PROGRAM Alarm
VAR
	Timer_allarme: TON;
	allarme_tamper:BOOL;
	Timer_Sirena: TP;
	alarm_service: BOOL;
	rilevato_movimento: BOOL;
	rilevata_manomissione: BOOL;
	allarme_scattato: BOOL;
	SR_ainterno: SR;
	SR_afronte: SR;
	SR_aretro: SR;
	SR_asx: SR;
	SR_allarme: SR;
	SR_atamper: SR;
	SR_mensa: SR;
	SR_ingresso: SR;
	SR_tecnico: SR;
	
	F1_trig: F_TRIG;
	F2_trig: F_TRIG;
	F3_trig: F_TRIG;
	F4_trig: F_TRIG;
	F5_trig: F_TRIG;
	S1_trig: F_TRIG;
	S2_trig: F_TRIG;
	R1_trig: F_TRIG;
	R2_trig: F_TRIG;
	R3_trig: F_TRIG;
	R4_trig: F_TRIG;
	R5_trig: F_TRIG;
	D1_trig: F_TRIG;
	C1_trig: F_TRIG;
	C2_trig: F_TRIG;
	C3_trig: F_TRIG;
	U1_trig: F_TRIG;
	U2_trig: F_TRIG;
	U3_trig: F_TRIG;

	F1_count: INT;
	F2_count: INT;
	F3_count: INT;
	F4_count: INT;
	F5_count: INT;
	S1_count: INT;
	S2_count: INT;
	R1_count: INT;
	R2_count: INT;
	R3_count: INT;
	R4_count: INT;
	R5_count: INT;
	D1_count: INT;
	C1_count: INT;
	C2_count: INT;
	C3_count: INT;
	U1_count: INT;
	U2_count: INT;
	U3_count: INT;
	radio_count: INT;
	sirena_count: INT;
	allarm_trig: R_TRIG;
	rtrig_radio: R_TRIG;
	rtrig_sirena: R_TRIG;
END_VAR

act();
(*Ritardo avvio allarme su accensione*)
//Timer_allarme(IN:= allarme, PT:= delay_allarme_on, Q=> allarme_on, ET=> );
(*Sensori*)
rilevato_movimento:=
	NOT (	
	SM_F1 AND
	SM_F2 AND
	SM_F3 AND
	SM_F4 AND
	SM_F5 AND
	SM_S1 AND
	SM_S2 AND
	//SM_R1 AND
	//SM_R2 AND
	//SM_R3 AND
	//SM_R4 AND
	//SM_R5 AND
	//SM_D1 AND
	SM_C1 AND
	//SM_C2 AND
	//SM_C3 AND
	SM_U1 AND 
	SM_U2 //AND
	//SM_U3 
	);
(*rilevata_manomissione:=NOT (Tamper_interno AND Tamper_fronte AND Tamper_retro AND Tamper_sinistro);*)
(*Ritardo spegnimento sirena*)
//Timer_Sirena(IN:= timer_Allarme.Q  AND rilevato_movimento, PT:= delay_sirena_off, Q=>, ET=> );
(*Azioni allarme*)
(*Segnale_sirena:=(timer_sirena.Q  AND NOT alarm_service) OR test_sirena;*)
//Segnale_radio:=(timer_sirena.Q AND NOT alarm_service) OR test_radio;
(*Allarme Tamper*)
allarme_tamper:=NOT alarm_service AND rilevata_manomissione;

IF allarme_Attivo<>0 (*allarme_on*) THEN
	//Gestione contatore sensore F1
	F1_trig(CLK:= SM_F1, Q=> );
	IF F1_trig.Q THEN
		F1_count:=F1_count+1;
	END_IF
	//Gestione contatore sensore F2
	F2_trig(CLK:= SM_F2, Q=> );
	IF F2_trig.Q THEN
		F2_count:=F2_count+1;
	END_IF
	//Gestione contatore sensore F3
	F3_trig(CLK:= SM_F3, Q=> );
	IF F3_trig.Q THEN
		F3_count:=F3_count+1;
	END_IF
	//Gestione contatore sensore F4
	F4_trig(CLK:= SM_F4, Q=> );
	IF F4_trig.Q THEN
		F4_count:=F4_count+1;
	END_IF
	//Gestione contatore sensore F5
	F5_trig(CLK:= SM_F5, Q=> );
	IF F5_trig.Q THEN
		F5_count:=F5_count+1;
	END_IF
	//Gestione contatore sensore S1
	S1_trig(CLK:= SM_S1, Q=> );
	IF S1_trig.Q THEN
		S1_count:=S1_count+1;
	END_IF
	//Gestione contatore sensore S2
	S2_trig(CLK:= SM_S2, Q=> );
	IF S2_trig.Q THEN
		S2_count:=S2_count+1;
	END_IF
	(*//Gestione contatore sensore R1
	R1_trig(CLK:= SM_R1, Q=> );
	IF R1_trig.Q THEN
		R1_count:=R1_count+1;
	END_IF
	//Gestione contatore sensore R2
	R2_trig(CLK:= SM_R2, Q=> );
	IF R2_trig.Q THEN
		R2_count:=R2_count+1;
	END_IF
	//Gestione contatore sensore R3
	R3_trig(CLK:= SM_R3, Q=> );
	IF R3_trig.Q THEN
		R3_count:=R3_count+1;
	END_IF
	//Gestione contatore sensore R4
	R4_trig(CLK:= SM_R4, Q=> );
	IF R4_trig.Q THEN
		R4_count:=R4_count+1;
	END_IF
	//Gestione contatore sensore R5
	R5_trig(CLK:= SM_R5, Q=> );
	IF R5_trig.Q THEN
		R5_count:=R5_count+1;
	END_IF
	//Gestione contatore sensore D1
	D1_trig(CLK:= SM_D1, Q=> );
	IF D1_trig.Q THEN
		D1_count:=D1_count+1;
	END_IF*)
	//Gestione contatore sensore C1
	C1_trig(CLK:= SM_C1, Q=> );
	IF C1_trig.Q THEN
		C1_count:=C1_count+1;
	END_IF
	(*//Gestione contatore sensore C2
	C2_trig(CLK:= SM_C2, Q=> );
	IF C2_trig.Q THEN
		C2_count:=C2_count+1;
	END_IF
	//Gestione contatore sensore C3
	C3_trig(CLK:= SM_C3, Q=> );
	IF C3_trig.Q THEN
		C3_count:=C3_count+1;
	END_IF*)
	//Gestione contatore sensore U1
	U1_trig(CLK:= SM_U1, Q=> );
	IF U1_trig.Q THEN
		U1_count:=U1_count+1;
	END_IF
	//Gestione contatore sensore U2
	U2_trig(CLK:= SM_U2, Q=> );
	IF U2_trig.Q THEN
		U2_count:=U2_count+1;
	END_IF
	(*//Gestione contatore sensore U3
	U3_trig(CLK:= SM_U3, Q=> );
	IF U3_trig.Q THEN
		U3_count:=U3_count+1;
	END_IF*)
	//Gestione contatore segnale radio e sirena
	rtrig_radio(CLK:= segnale_radio, Q=> );
	rtrig_sirena(CLK:= segnale_sirena, Q=> );
	IF rtrig_radio.Q THEN
		radio_count:=radio_count+1;
	END_IF
	IF rtrig_sirena.Q THEN
		sirena_count:=sirena_count+1;
	END_IF
END_IF
allarm_trig(CLK:= allarme_Attivo<>0 (*allarme*), Q=> );
IF allarm_trig.Q THEN
	F1_count:=0;
	F2_count:=0;
	F3_count:=0;
	F4_count:=0;
	F5_count:=0;
	S1_count:=0;
	S2_count:=0;
	R1_count:=0;
	R2_count:=0;
	R3_count:=0;
	R4_count:=0;
	R5_count:=0;
	D1_count:=0;
	C1_count:=0;
	C2_count:=0;
	C3_count:=0;
	U1_count:=0;
	U2_count:=0;
	U3_count:=0;
	radio_count:=0;
	sirena_count:=0;
END_IF
//Gestione sensori movimento
sensori_STRU[0](indice:=0); //Sensore movimento frontale 1
sensori_STRU[1](indice:=1); //Sensore movimento frontale 2
sensori_STRU[2](indice:=2); //Sensore movimento frontale 3
sensori_STRU[3](indice:=3); //Sensore movimento frontale 4
sensori_STRU[4](indice:=4); //Sensore movimento frontale 5
sensori_STRU[5](indice:=5); //Sensore movimento sinistro 1
sensori_STRU[6](indice:=6); //Sensore movimento sinistro 2
sensori_STRU[7](indice:=7); //Sensore movimento retro 1
sensori_STRU[8](indice:=8); //Sensore movimento retro 2
sensori_STRU[9](indice:=9); //Sensore movimento retro 3
sensori_STRU[10](indice:=10); //Sensore movimento retro 4
sensori_STRU[11](indice:=11); //Sensore movimento retro 5
sensori_STRU[12](indice:=12); //Sensore movimento destro
sensori_STRU[13](indice:=13); //Sensore movimento centrale 1
sensori_STRU[14](indice:=14); //Sensore movimento centrale 2
sensori_STRU[15](indice:=15); //Sensore movimento centrale 3
sensori_STRU[16](indice:=16); //Sensore movimento ufficio tecnico U1
sensori_STRU[17](indice:=17); //Sensore movimento locale svago U2
sensori_STRU[18](indice:=18); //Sensore movimento ingresso U3

//Attivazione segnale sirena-radio allarme
IF ((sens_allarme_Stru[0].allarme_sensore OR 
	sens_allarme_stru[1].allarme_sensore OR
	sens_allarme_Stru[2].allarme_sensore OR
	sens_allarme_stru[3].allarme_sensore OR
	sens_Allarme_stru[4].allarme_sensore OR
	sens_allarme_stru[5].allarme_sensore OR
	sens_allarme_Stru[6].allarme_sensore OR
	sens_allarme_stru[13].allarme_sensore OR
	sens_allarme_Stru[16].allarme_sensore OR
	sens_allarme_Stru[17].allarme_sensore) AND NOT alarm_Service) THEN
		allarme_scattato:=TRUE;
ELSE
		allarme_scattato:=FALSE;
END_IF
segnale_sirena:=(allarme_Scattato AND HMI_sirena) OR test_sirena;	
segnale_radio:=(allarme_scattato AND HMI_radio) OR test_radio;
ingresso_sens[0]:=SM_F1;
ingresso_sens[1]:=SM_F2;
ingresso_sens[2]:=SM_F3;
ingresso_sens[3]:=SM_F4;
ingresso_sens[4]:=SM_F5;
ingresso_sens[5]:=SM_S1;
ingresso_sens[6]:=SM_S2;
ingresso_sens[13]:=SM_C1;
ingresso_sens[16]:=SM_U1;
ingresso_sens[17]:=SM_U2;

ACTION ACT:
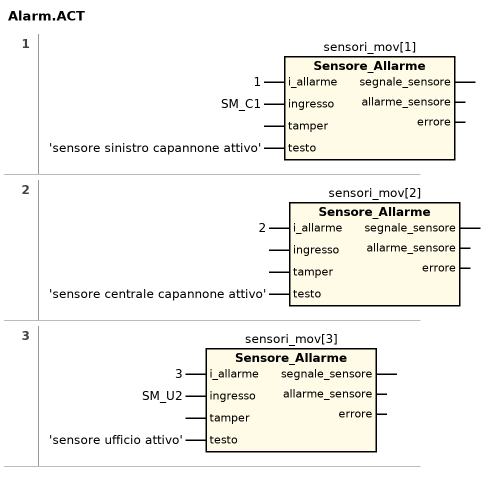
// NETWORK 1
sensori_mov[1](i_allarme := 1, ingresso := SM_C1, testo := 'sensore sinistro capannone attivo'); // Sensore_Allarme

// NETWORK 2
sensori_mov[2](i_allarme := 2, testo := 'sensore centrale capannone attivo'); // Sensore_Allarme

// NETWORK 3
sensori_mov[3](i_allarme := 3, ingresso := SM_U2, testo := 'sensore ufficio attivo'); // Sensore_Allarme
END_ACTION

END_PROGRAM

(* stored: Version 1.1.0.1, ProductVersion 3.1.4022.18
   POU Alarm: Id {1fb85a97-8a0b-451f-b10d-e0cebcbc9d7e}, SpecialFunc None
   Action ACT: Id {1e07d8a0-35d1-4acd-9022-39fc95565760} *)
